(* PLC project Unnamed, Unknown Unnamed 1 *)
(* stored: creationDateTime 2019-11-03T20:00:54, modificationDateTime 2019-12-11T16:49:48 *)

PROGRAM program0
  VAR
    van1 AT %QX100.0 : BOOL;  (* 800 *)
    quat1 AT %QX100.1 : BOOL;  (* 801 *)
    den1 AT %QX100.2 : BOOL;  (* 802 *)
    van2 AT %QX100.3 : BOOL;  (* 803 *)
    quat2 AT %QX100.4 : BOOL;  (* 804 *)
    den2 AT %QX100.5 : BOOL;  (* 805 *)
    cambien1 AT %IW100 : UINT;  (* 100 *)
    cambien2 AT %IW101 : UINT;  (* 101 *)
    set_nhietdo AT %MW7 : UINT;  (* 1031 *)
    set_doam AT %MW8 : UINT;  (* 1032 *)
    set_van1 AT %MW1 : UINT;  (* 1025 *)
    set_manual AT %MW9 : UINT;  (* 1033 *)
    set_van2 AT %MW2 : UINT;  (* 1026 *)
    set_den1 AT %MW3 : UINT;  (* 1027 *)
    set_den2 AT %MW4 : UINT;  (* 1028 *)
    set_quat1 AT %MW5 : UINT;  (* 1029 *)
    set_quat2 AT %MW6 : UINT;  (* 1030 *)
  END_VAR
  VAR_TEMP
    temp_manual : BOOL;
    temp_van1 : BOOL;
    temp_van2 : BOOL;
    temp_den1 : BOOL;
    temp_den2 : BOOL;
    temp_quat1 : BOOL;
    temp_quat2 : BOOL;
    temp_nhietdo : BOOL;
    temp_doam : BOOL;
    temp_MUL_nhietdo : UINT;
    temp_cambien2_udint : UDINT;
    temp_MUL_doam : UDINT;
  END_VAR
  VAR
    result_nhietdo AT %MW10 : UINT;  (* 1034 *)
    result_doam AT %MW11 : UINT;  (* 1035 *)
  END_VAR
  VAR_TEMP
    temp_result_doam_udint : UDINT;
  END_VAR
  VAR
    time_bat_den AT %MW12 : UINT;  (* 1036 *)
  END_VAR
  VAR_TEMP
    temp_time_bat_den : TIME;
    temp_time_bat_den_delay : TIME;
  END_VAR
  VAR
    time_bat_den_delay AT %MW13 : UINT;  (* 1037 *)
  END_VAR
  VAR_TEMP
    temp_start_stop : BOOL;
  END_VAR
  VAR
    start_stop AT %MW14 : UINT;  (* 1038 *)
  END_VAR
  VAR
    TON0 : TON;
    TON1 : TON;
    temp_on1 : BOOL;
    temp_on0 : BOOL;
  END_VAR

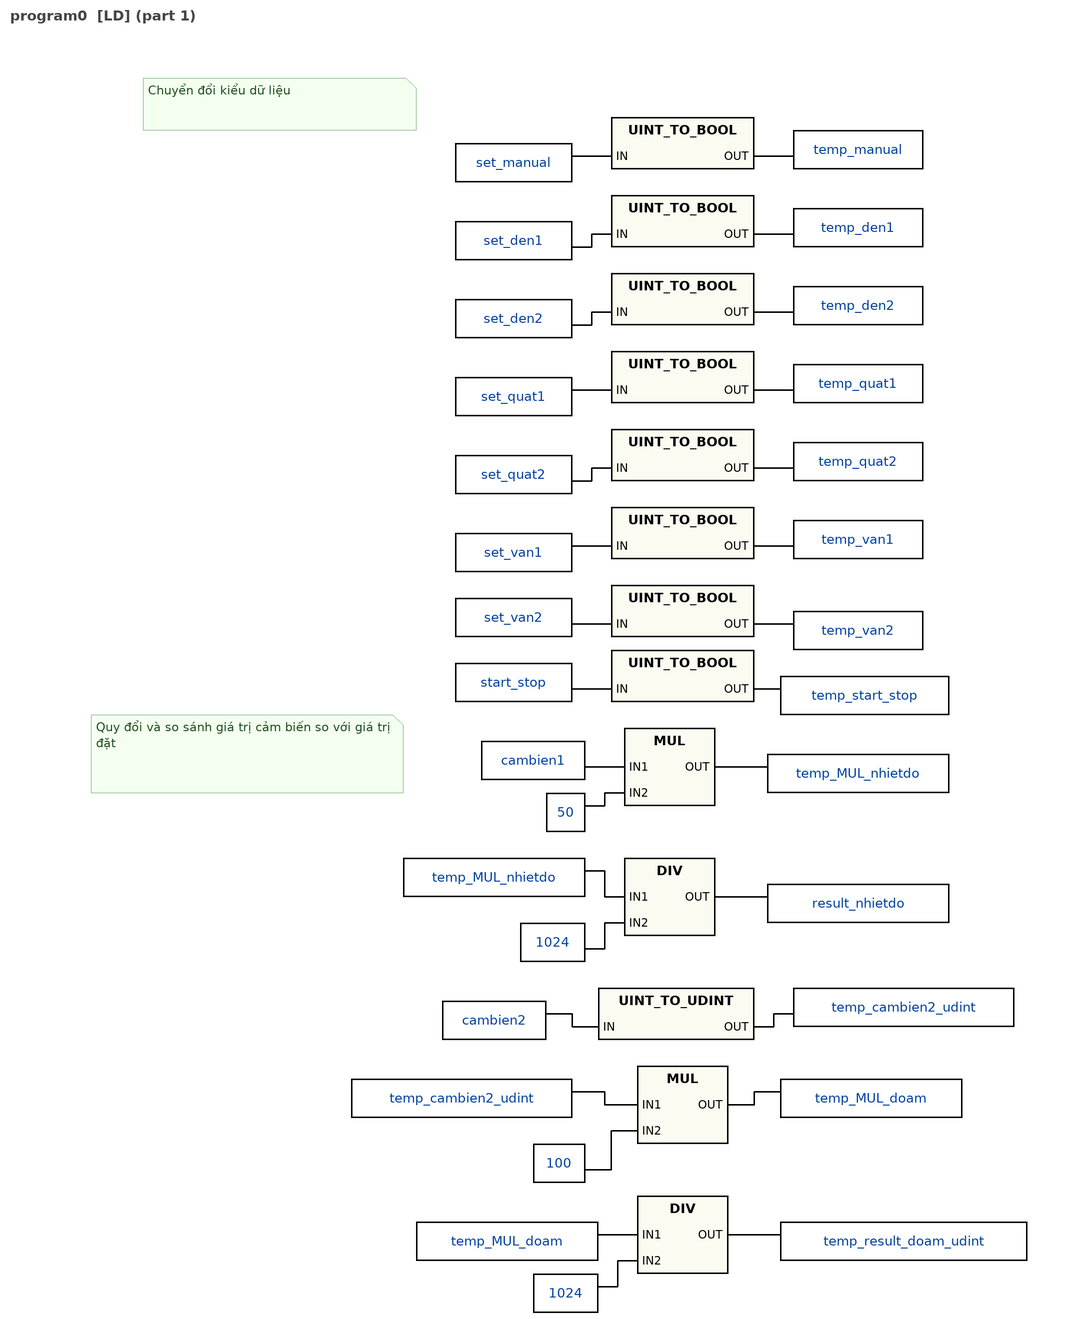
(* LD diagram, written out as Structured Text *)
(* Chuyển đổi kiểu dữ liệu *)
temp_manual := UINT_TO_BOOL(set_manual);
temp_den1 := UINT_TO_BOOL(set_den1);
temp_den2 := UINT_TO_BOOL(set_den2);
temp_quat1 := UINT_TO_BOOL(set_quat1);
temp_quat2 := UINT_TO_BOOL(set_quat2);
temp_van1 := UINT_TO_BOOL(set_van1);
temp_van2 := UINT_TO_BOOL(set_van2);
temp_start_stop := UINT_TO_BOOL(start_stop);
(* Quy đổi và so sánh giá trị cảm biến so với giá trị đặt *)
temp_MUL_nhietdo := cambien1 * 50;
result_nhietdo := temp_MUL_nhietdo / 1024;
temp_cambien2_udint := UINT_TO_UDINT(cambien2);
temp_MUL_doam := temp_cambien2_udint * 100;
temp_result_doam_udint := temp_MUL_doam / 1024;
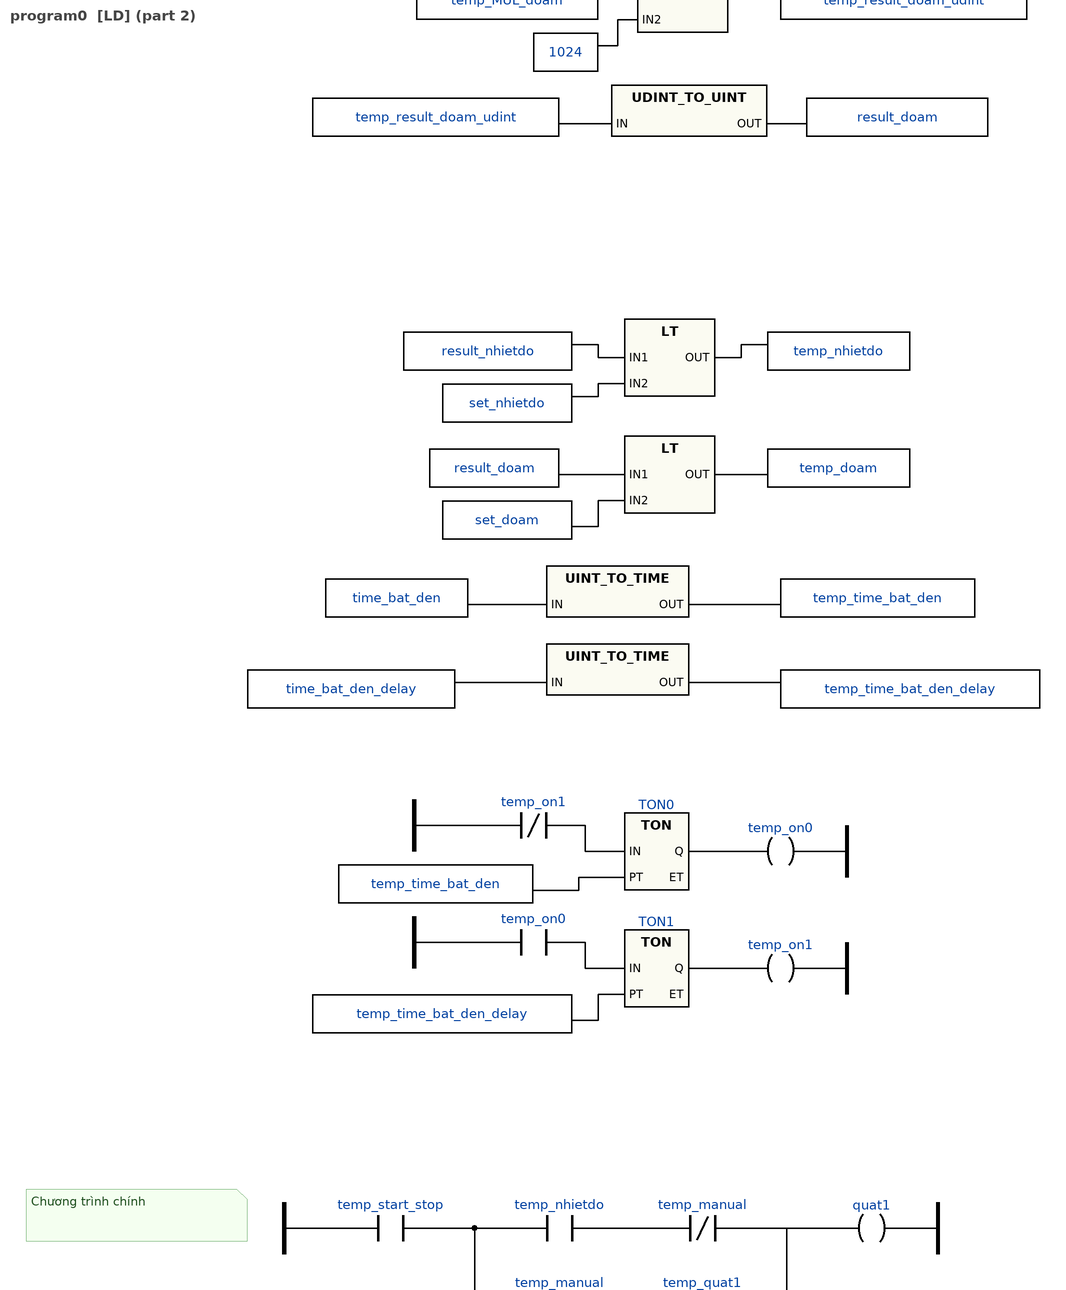
result_doam := UDINT_TO_UINT(temp_result_doam_udint);
temp_nhietdo := result_nhietdo < set_nhietdo;
temp_doam := result_doam < set_doam;
temp_time_bat_den := UINT_TO_TIME(time_bat_den);
temp_time_bat_den_delay := UINT_TO_TIME(time_bat_den_delay);
TON0(IN := NOT temp_on1, PT := temp_time_bat_den);
temp_on0 := TON0.Q;
TON1(IN := temp_on0, PT := temp_time_bat_den_delay);
temp_on1 := TON1.Q;
(* Chương trình chính *)
quat1 := temp_start_stop AND (temp_nhietdo AND NOT temp_manual OR temp_manual AND temp_quat1);
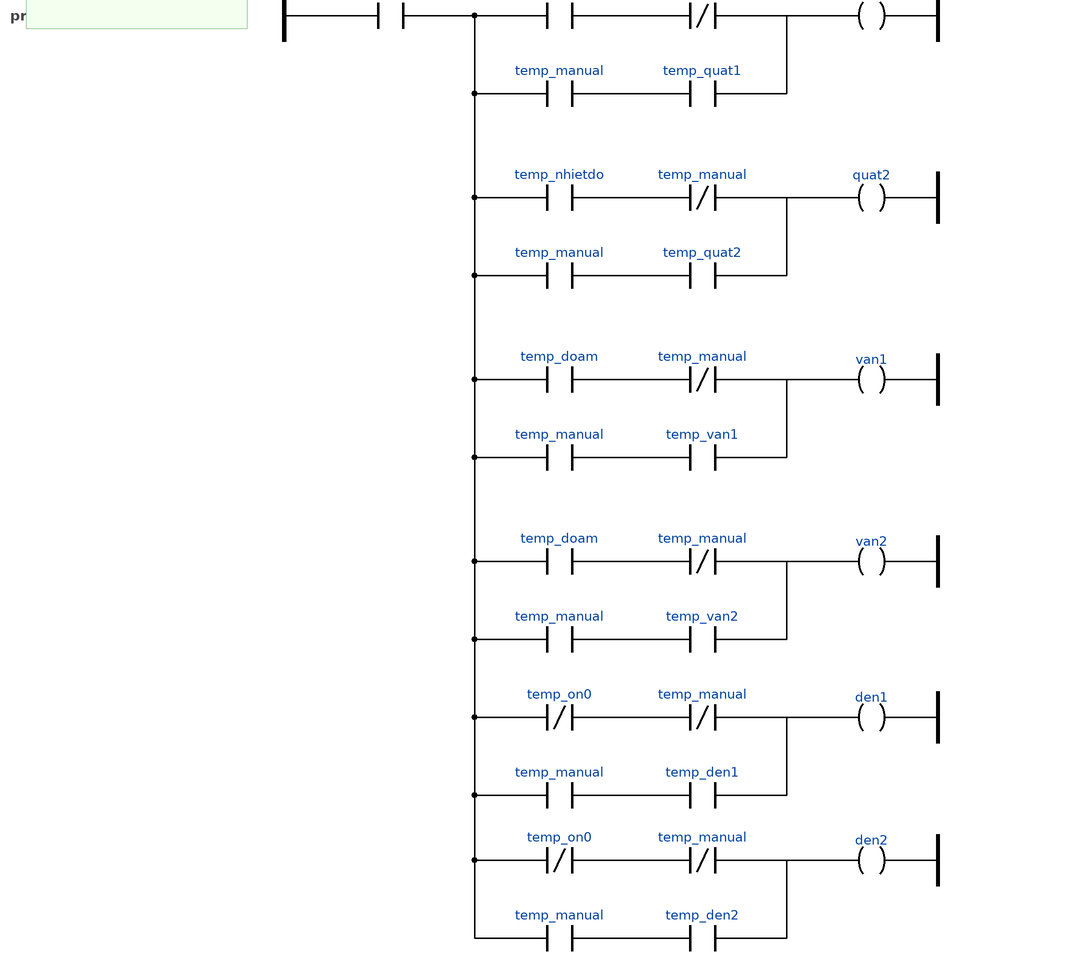
quat2 := temp_start_stop AND (temp_nhietdo AND NOT temp_manual OR temp_manual AND temp_quat2);
van1 := temp_start_stop AND (temp_doam AND NOT temp_manual OR temp_manual AND temp_van1);
van2 := temp_start_stop AND (temp_doam AND NOT temp_manual OR temp_manual AND temp_van2);
den1 := temp_start_stop AND (NOT temp_on0 AND NOT temp_manual OR temp_manual AND temp_den1);
den2 := temp_start_stop AND (NOT temp_on0 AND NOT temp_manual OR temp_manual AND temp_den2);
END_PROGRAM

CONFIGURATION Config0
  RESOURCE Res0 ON PLC
    TASK task0(INTERVAL := T#20ms, PRIORITY := 0);
    PROGRAM instance0 WITH task0 : program0;
  END_RESOURCE
END_CONFIGURATION
